FUNCTION_BLOCK FB_FeedMeina2_750x750_Circles EXTENDS FB_RecipeBase

METHOD Build : BOOL
VAR
    TotalX, TotalY, Radius : LREAL;
    CircleRadius           : LREAL;
    Velo                   : LREAL;
    localConfig            : ST_GantryXYZ_Config;
    
    PanelGap               : LREAL;
    Y_Offset               : LREAL;
    p                      : INT;

    HoleDistanceFromEdgeOfRail : LREAL := 100.0;
    SomeFixedDimension         : LREAL := 12.63;
    PanelRailOffsetX           : LREAL;
    PanelRailOffsetY           : LREAL;
    ExtrusionLengthX           : LREAL;
    ExtrusionLengthY           : LREAL;
    
    NumberOfHolesX             : INT := 3;
    NumberOfHolesY             : INT := 5;
    HolesSpacingX              : LREAL;
    HolesSpacingY              : LREAL;
    
    i                          : INT;
    holeIdx                    : INT;
    
    RailSlot  : LREAL := 29.0;
    BigSlot   : LREAL := 200.0;
    SmallSlot : LREAL := 100.0;

    LeadInY   : LREAL := 10.0;
    LeadOutY  : LREAL := 10.0;

    sx : LREAL;
    sy : LREAL;
    dx : LREAL;
    dy : LREAL;
    r_val : LREAL;
END_VAR
_Busy := TRUE;
_Done := FALSE;
_Error := FALSE;
Build := FALSE;
THIS^.UpdateNestingLimits();

IF NOT _Config.IsValid THEN
    _Busy := FALSE;
    _Error := TRUE; 
    Build := FALSE;
    RETURN;
END_IF

// Zmiana rozmiaru na 750mm
TotalX := 750.0;
TotalY := 750.0;
CircleRadius := TotalX / 2.0;

PanelGap := 20.0; 

PanelRailOffsetX := 0.1 * TotalX;
PanelRailOffsetY := 0.1 * TotalY;

ExtrusionLengthX := TotalX - (2.0 * PanelRailOffsetX);
ExtrusionLengthY := TotalY - (2.0 * PanelRailOffsetY);

IF NumberOfHolesX > 1 THEN
    HolesSpacingX := (ExtrusionLengthX - (2.0 * HoleDistanceFromEdgeOfRail)) / INT_TO_LREAL(NumberOfHolesX - 1);
ELSE
    HolesSpacingX := 0.0;
END_IF

IF NumberOfHolesY > 1 THEN
    HolesSpacingY := (ExtrusionLengthY - (2.0 * HoleDistanceFromEdgeOfRail)) / INT_TO_LREAL(NumberOfHolesY - 1);
ELSE
    HolesSpacingY := 0.0;
END_IF

holeIdx := 0; 

// Pętla zmieniona na 3 elementy (0 DO 2)
FOR p := 0 TO 2 DO
    Y_Offset := INT_TO_LREAL(p) * (TotalY + PanelGap);

    holeIdx := holeIdx + 1;
    _HolesDrill[holeIdx].X := LREAL_TO_REAL(TotalX / 2.0);
    _HolesDrill[holeIdx].Y := LREAL_TO_REAL((TotalY / 2.0) + Y_Offset);

    FOR i := NumberOfHolesY TO 1 BY -1 DO
        holeIdx := holeIdx + 1;
        _HolesDrill[holeIdx].X := LREAL_TO_REAL(PanelRailOffsetX - SomeFixedDimension);
        _HolesDrill[holeIdx].Y := LREAL_TO_REAL(PanelRailOffsetY + HoleDistanceFromEdgeOfRail + ((i - 1) * HolesSpacingY) + Y_Offset);
    END_FOR

    FOR i := 1 TO NumberOfHolesX DO
        holeIdx := holeIdx + 1;
        _HolesDrill[holeIdx].X := LREAL_TO_REAL(PanelRailOffsetX + HoleDistanceFromEdgeOfRail + ((i - 1) * HolesSpacingX));
        _HolesDrill[holeIdx].Y := LREAL_TO_REAL(PanelRailOffsetY - SomeFixedDimension + Y_Offset);
    END_FOR

    FOR i := 1 TO NumberOfHolesY DO
        holeIdx := holeIdx + 1;
        _HolesDrill[holeIdx].X := LREAL_TO_REAL(PanelRailOffsetX + ExtrusionLengthX + SomeFixedDimension);
        _HolesDrill[holeIdx].Y := LREAL_TO_REAL(PanelRailOffsetY + HoleDistanceFromEdgeOfRail + ((i - 1) * HolesSpacingY) + Y_Offset);
    END_FOR

    FOR i := NumberOfHolesX TO 1 BY -1 DO
        holeIdx := holeIdx + 1;
        _HolesDrill[holeIdx].X := LREAL_TO_REAL(PanelRailOffsetX + HoleDistanceFromEdgeOfRail + ((i - 1) * HolesSpacingX));
        _HolesDrill[holeIdx].Y := LREAL_TO_REAL(PanelRailOffsetY + ExtrusionLengthY + SomeFixedDimension + Y_Offset);
    END_FOR
END_FOR

_HolesToDrill := holeIdx;

// Liczba kształtów to teraz 8 (3 kółka + 5 dotychczasowych profili/otworów)
_ShapesCount := 8; 

// Kółko 1
_ShapeStart[1].X := TotalX;
_ShapeStart[1].Y := CircleRadius - LeadInY;

// Kółko 2
_ShapeStart[2].X := TotalX;
_ShapeStart[2].Y := TotalY + PanelGap + CircleRadius - LeadInY;

// Kółko 3
_ShapeStart[3].X := TotalX;
_ShapeStart[3].Y := 2.0 * (TotalY + PanelGap) + CircleRadius - LeadInY;

// Pozostałe kształty przesunięte na indeksy 4-8 
// UWAGA: Stałe współrzędne > 750 (np. 900.0) mogą wymagać Twojej poprawki do nowego wymiaru TotalX/Y
_ShapeStart[4].X := 900.0;
_ShapeStart[4].Y := 125.0;

_ShapeStart[5].X := 900.0;
_ShapeStart[5].Y := 875.0;

_ShapeStart[6].X := 920.0;
_ShapeStart[6].Y := 20.0;

_ShapeStart[7].X := 870.0;
_ShapeStart[7].Y := 220.0;

_ShapeStart[8].X := 870.0;
_ShapeStart[8].Y := 520.0;

IF _ConfigProvider <> 0 THEN
    localConfig := _ConfigProvider.Config;
    Velo := localConfig.CuttingSpeedXY;
ELSE
    Velo := 50.0;
END_IF

_GeometryWriter.Clear();
_GeometryWriter.EnableTangentialFollowing();

sx := 0.0; sy := 0.0; dx := 0.0; dy := 0.0; r_val := 0.0;

CASE _CurrentShapeIndex OF
    // Obsługa cięcia 3 kółek w ten sam sposób
    1, 2, 3:
        Y_Offset := INT_TO_LREAL(_CurrentShapeIndex - 1) * (TotalY + PanelGap);

        _GeometryWriter.AddStartPoint(_ShapeStart[_CurrentShapeIndex].X, _ShapeStart[_CurrentShapeIndex].Y); 
        _GeometryWriter.AddLine(TotalX, CircleRadius + Y_Offset, Velo); 
        _GeometryWriter.AddArc(0.0, CircleRadius + Y_Offset, CircleRadius, CircleRadius + Y_Offset, Velo, FALSE);
        _GeometryWriter.AddArc(TotalX, CircleRadius + Y_Offset, CircleRadius, CircleRadius + Y_Offset, Velo, FALSE);
        _GeometryWriter.AddLine(TotalX, CircleRadius + LeadOutY + Y_Offset, Velo); 

    // Obsługa pozostałych wycięć
    4, 5, 6, 7, 8:
        sx := _ShapeStart[_CurrentShapeIndex].X;
        sy := _ShapeStart[_CurrentShapeIndex].Y;
        r_val := 10.0;

        IF _CurrentShapeIndex = 4 THEN
            dx := RailSlot;
            dy := ExtrusionLengthY;
        ELSIF _CurrentShapeIndex = 5 THEN
            dx := RailSlot;
            dy := ExtrusionLengthX; 
        ELSIF _CurrentShapeIndex = 6 THEN
            dx := SmallSlot;
            dy := SmallSlot;
        ELSIF _CurrentShapeIndex = 7 THEN
            dx := BigSlot;
            dy := BigSlot;
        ELSIF _CurrentShapeIndex = 8 THEN
            dx := BigSlot;
            dy := BigSlot;
        END_IF

        _GeometryWriter.AddStartPoint(sx, sy);

        _GeometryWriter.AddLine(sx, sy + dy - r_val, Velo);
        IF r_val > 0 THEN
            _GeometryWriter.AddArc(sx + r_val, sy + dy, sx + r_val, sy + dy - r_val, Velo, TRUE);
        END_IF

        _GeometryWriter.AddLine(sx + dx - r_val, sy + dy, Velo);
        IF r_val > 0 THEN
            _GeometryWriter.AddArc(sx + dx, sy + dy - r_val, sx + dx - r_val, sy + dy - r_val, Velo, TRUE);
        END_IF

        _GeometryWriter.AddLine(sx + dx, sy + r_val, Velo);
        IF r_val > 0 THEN
            _GeometryWriter.AddArc(sx + dx - r_val, sy, sx + dx - r_val, sy + r_val, Velo, TRUE);
        END_IF

        _GeometryWriter.AddLine(sx + r_val, sy, Velo);
        IF r_val > 0 THEN
            _GeometryWriter.AddArc(sx, sy + r_val, sx + r_val, sy + r_val, Velo, TRUE);
        END_IF

END_CASE

_GeometryWriter.EndTable();

_Busy := FALSE;
_Done := TRUE;
Build := TRUE;
END_METHOD

METHOD PROTECTED CalculateFootprint
VAR_INPUT
END_VAR
_NominalX := 1200;
_NominalY := 2400;
END_METHOD

PROPERTY ExecutionRoute : E_ExecutionRoute
GET
ExecutionRoute := E_ExecutionRoute.eFeedTable;
END_GET
END_PROPERTY

METHOD FB_init : BOOL
VAR_INPUT
	bInitRetains : BOOL; // if TRUE, the retain variables are initialized (warm start / cold start)
	bInCopyCode : BOOL;  // if TRUE, the instance afterwards gets moved into the copy code (online change)
END_VAR
_Limits.PanelFrontLength.MinVal := 100.0;
_Limits.PanelFrontLength.MaxVal := 2400.0;

_Limits.PanelFrontWidth.MinVal  := 100.0;
_Limits.PanelFrontWidth.MaxVal  := 1200.0;

_Limits.PanelHeight.MinVal      := 0.0;
_Limits.PanelHeight.MaxVal      := 0.0;

_Limits.RailHeightCorrection.MinVal := 0.0;
_Limits.RailHeightCorrection.MaxVal := 0.0;

_Limits.CuttingOverpass.MinVal := 0.0;
_Limits.CuttingOverpass.MaxVal := 50.0;

_Limits.GroovingOverpass.MinVal := 0.0;
_Limits.GroovingOverpass.MaxVal := 50.0;

_Limits.GrooveDepthZ.MinVal := 0.0;
_Limits.GrooveDepthZ.MaxVal := 9.0; 

_Limits.CuttingOverpass.MinVal := 0.0;
_Limits.CuttingOverpass.MaxVal := 50.0;
_Limits.GroovingOverpass.MinVal := 0.0;
_Limits.GroovingOverpass.MaxVal := 50.0;

_Limits.Radius.MinVal := 10.0;     
_Limits.Radius.MaxVal := 600.0;
END_METHOD

END_FUNCTION_BLOCK

(* stored: Version 1.1.0.1, ProductVersion 3.1.4024.15
   POU FB_FeedMeina2_750x750_Circles: Id {10bc1678-2212-4f03-9d76-3e10f94eddda}, SpecialFunc None
   Method Build: Id {9afe5b79-08bb-4ebd-8601-9ec8c62c93f9}
   Method CalculateFootprint: Id {3574da9d-4b8a-441e-a2e2-40ddce951262}
   Property ExecutionRoute: Id {02397026-5ced-429c-aa50-9358e8b3594b}
   Get Get: Id {de57a927-834e-4101-9c42-8d78ea7f5d4b}
   Method FB_init: Id {8165bd51-d856-4c63-95fe-7f71907d18f8} *)
